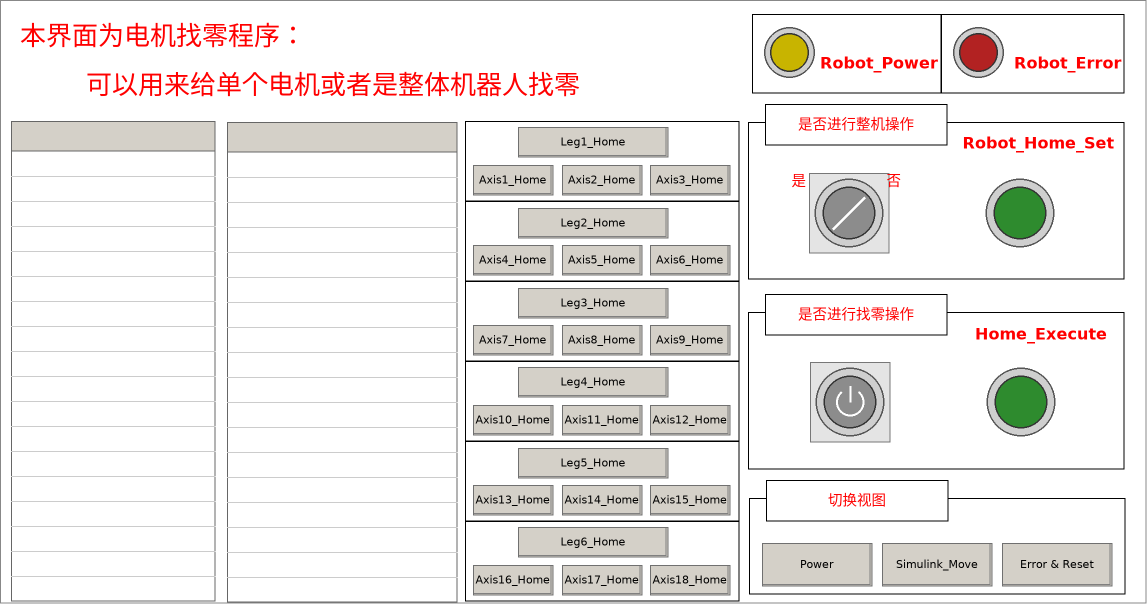
VISUALIZATION Visu_Home  // 1147x604
    Rectangle (752,14 189x79)
    Rectangle (748,312 376x157)
    Label (964,318 154x32), "Home_Execute"
    Rectangle (765,294 182x41), "是否进行找零操作"
    Lamp1 (981,362 80x80), variable: Home_Execute, style: Lamp-Lamp1-Green
    PowerSwitch (810,362 80x80), variable: Home_Execute, behaviour: TOGGLE, style: Switch-PowerSwitch-Gray
    Rectangle (941,14 183x79)
    Lamp1 (948,23 61x59), variable: Hexapod_Robot.Robot_Error, style: Lamp-Lamp1-Red
    Label (991,47 154x32), "Robot_Error"
    Label (17,15 365x42), "本界面为电机找零程序："
    Label (83,64 874x42), "可以用来给单个电机或者是整体机器人找零"
    Table (11,121 204x480), data array: Hexapod_Robot.Axis_ActPostion
        p3854506369: Hexapod_Robot.Axis_ActPostion[INDEX]
        p2232123230: Axis_ActPostion[Robot]
    Table (227,122 230x480), data array: Hexapod_Robot.Current_Turque_Value
        p3854506369: Hexapod_Robot.Current_Turque_Value[INDEX]
        p2232123230: Current_Turque_Value[Robot]
    Lamp1 (759,23 61x59), variable: Hexapod_Robot.Robot_Power, style: Lamp-Lamp1-Yellow
    Label (802,47 154x32), "Robot_Power"
    Rectangle (465,121 274x80)
    Button (473,165 80x30), "Axis1_Home"
        toggle Hexapod_Robot.Axis_Home_Set[1]
        OnMouseClick: change screen: Visu_Home
    Button (650,165 80x30), "Axis3_Home"
        toggle Hexapod_Robot.Axis_Home_Set[3]
        OnMouseClick: change screen: Visu_Home
    Button (562,165 80x30), "Axis2_Home"
        toggle Hexapod_Robot.Axis_Home_Set[2]
        OnMouseClick: change screen: Visu_Home
    Rectangle (465,201 274x80)
    Button (473,245 80x30), "Axis4_Home"
        toggle Hexapod_Robot.Axis_Home_Set[4]
        OnMouseClick: change screen: Visu_Home
    Button (650,245 80x30), "Axis6_Home"
        toggle Hexapod_Robot.Axis_Home_Set[6]
        OnMouseClick: change screen: Visu_Home
    Button (562,245 80x30), "Axis5_Home"
        toggle Hexapod_Robot.Axis_Home_Set[5]
        OnMouseClick: change screen: Visu_Home
    Rectangle (465,281 274x80)
    Button (473,325 80x30), "Axis7_Home"
        toggle Hexapod_Robot.Axis_Home_Set[7]
        OnMouseClick: change screen: Visu_Home
    Button (650,325 80x30), "Axis9_Home"
        toggle Hexapod_Robot.Axis_Home_Set[9]
        OnMouseClick: change screen: Visu_Home
    Button (562,325 80x30), "Axis8_Home"
        toggle Hexapod_Robot.Axis_Home_Set[8]
        OnMouseClick: change screen: Visu_Home
    Rectangle (465,361 274x80)
    Button (473,405 80x30), "Axis10_Home"
        toggle Hexapod_Robot.Axis_Home_Set[10]
        OnMouseClick: change screen: Visu_Home
    Button (650,405 80x30), "Axis12_Home"
        toggle Hexapod_Robot.Axis_Home_Set[12]
        OnMouseClick: change screen: Visu_Home
    Button (562,405 80x30), "Axis11_Home"
        toggle Hexapod_Robot.Axis_Home_Set[11]
        OnMouseClick: change screen: Visu_Home
    Rectangle (465,441 274x80)
    Button (473,485 80x30), "Axis13_Home"
        toggle Hexapod_Robot.Axis_Home_Set[13]
        OnMouseClick: change screen: Visu_Home
    Button (650,485 80x30), "Axis15_Home"
        toggle Hexapod_Robot.Axis_Home_Set[15]
        OnMouseClick: change screen: Visu_Home
    Button (562,485 80x30), "Axis14_Home"
        toggle Hexapod_Robot.Axis_Home_Set[14]
        OnMouseClick: change screen: Visu_Home
    Rectangle (465,521 274x80)
    Button (473,565 80x30), "Axis16_Home"
        toggle Hexapod_Robot.Axis_Home_Set[16]
        OnMouseClick: change screen: Visu_Home
    Button (650,565 80x30), "Axis18_Home"
        toggle Hexapod_Robot.Axis_Home_Set[18]
        OnMouseClick: change screen: Visu_Home
    Button (562,565 80x30), "Axis17_Home"
        toggle Hexapod_Robot.Axis_Home_Set[17]
        OnMouseClick: change screen: Visu_Home
    Rectangle (749,498 376x96)
    Rectangle (766,480 182x41), "切换视图"
    Button (762,543 110x43), "Power"
        OnMouseClick: change screen: Visu_Power
    Button (1002,543 110x43), "Error & Reset"
        OnMouseClick: change screen: Visu_Reset
    Button (882,543 110x43), "Simulink_Move"
        OnMouseClick: change screen: Visu_SimulinkMove
    Rectangle (748,122 376x157)
    Rectangle (765,104 182x41), "是否进行整机操作"
    Lamp1 (980,173 80x80), variable: Hexapod_Robot.Robot_Home_Set, style: Lamp-Lamp1-Green
    RotarySwitch (809,173 80x80), variable: Hexapod_Robot.Robot_Home_Set, behaviour: TOGGLE, style: Switch-RotarySwitch-Gray
    Label (864,166 60x30), "否"
    Label (769,166 60x30), "是"
    Label (935,127 207x32), "Robot_Home_Set"
    Button (518,127 150x30), "Leg1_Home"
        tap Hexapod_Robot.Leg_Home_Set[1]
    Button (518,208 150x30), "Leg2_Home"
        tap Hexapod_Robot.Leg_Home_Set[2]
    Button (518,288 150x30), "Leg3_Home"
        tap Hexapod_Robot.Leg_Home_Set[3]
    Button (518,367 150x30), "Leg4_Home"
        tap Hexapod_Robot.Leg_Home_Set[4]
    Button (518,448 150x30), "Leg5_Home"
        tap Hexapod_Robot.Leg_Home_Set[5]
    Button (518,527 150x30), "Leg6_Home"
        tap Hexapod_Robot.Leg_Home_Set[6]
END_VISUALIZATION

(* stored: Version 1.1.0.1, ProductVersion 3.1.4020.12
   Visu Visu_Home: Id {f1fd6469-4ee4-4390-8668-28dd879e70aa} *)
